PROGRAM MAIN
VAR
	MaquinaLigada: BOOL;
	bHabilita: BOOL;
	fb_Habilita1: MC_Power;
END_VAR

//Ler Status
	Eixos.Eixo1.ReadStatus();
	Eixos.Eixo2.ReadStatus();
	
//Habilitar Eixo1
IF MaquinaLigada THEN
		bHabilita := 1;
	ELSE
		bHabilita := 0;
	END_IF
	fb_Habilita1(
		Axis:= Eixos.Eixo1, 
		Enable:= bHabilita, 
		Enable_Positive:= bHabilita, 
		Enable_Negative:= bHabilita, 
		Override:= 100.0);

END_PROGRAM

(* stored: Version 1.1.0.1, ProductVersion 3.1.4024.13
   POU MAIN: Id {91b9bb0d-f515-449b-b56e-1605f4f5713d}, SpecialFunc None *)
